(* PLC project PLC107_AO, home PLC107_AO 1 *)
(* stored: creationDateTime 2019-11-13T09:37:45, productRelease 0, modificationDateTime 2020-07-16T10:40:43, version 1 *)

(* Установка режима работы аналогового выхода *)
FUNCTION_BLOCK AOMode
  VAR_INPUT
    Ex : BOOL := FALSE;  (* разрешение на выполнение *)
    AOn : BYTE := 0;  (* номер выхода *)
    M : BYTE := 0;  (* режим работы *)
  END_VAR
  VAR_OUTPUT
    Om : BYTE := 0;  (* режим работы (установленный) *)
    Ok : BYTE := 0;  (* код результата исполнения блока *)
  END_VAR

            {extern void App_AOMode(AOMODE*);App_AOMode(data__);}

          
END_FUNCTION_BLOCK

(* Установка значения нормального аналогового выхода *)
FUNCTION_BLOCK AOVal
  VAR_INPUT
    Ex : BOOL := FALSE;  (* разрешение на выполнение *)
    AOn : BYTE := 0;  (* номер выхода *)
    V : REAL := 0.0;  (* значение *)
  END_VAR
  VAR_OUTPUT
    Ov : REAL := 0.0;  (* значение (установленное) *)
    Ok : BYTE := 0;  (* код результата исполнения блока *)
  END_VAR

            {extern void App_AOVal(AOVAL*);App_AOVal(data__);}

          
END_FUNCTION_BLOCK

(* Установка значения быстрого аналогового выхода *)
FUNCTION_BLOCK AOFast
  VAR_INPUT
    Ex : BOOL := FALSE;  (* разрешение на выполнение *)
    AOn : BYTE := 0;  (* номер выхода *)
    V : REAL := 0.0;  (* значение быстрого выхода *)
  END_VAR
  VAR_OUTPUT
    Ov : REAL := 0.0;  (* значение быстрого выхода (установленное) *)
    Ok : BYTE := 0;  (* код результата исполнения блока *)
  END_VAR

            {extern void App_AOFast(AOFAST*);App_AOFast(data__);}

          
END_FUNCTION_BLOCK

(* Установка безопасного значения аналогового выхода *)
FUNCTION_BLOCK AOSafe
  VAR_INPUT
    Ex : BOOL := FALSE;  (* разрешение на выполнение *)
    Enx : BOOL := FALSE;  (* разрешение быстрого выхода *)
    AOn : BYTE := 0;  (* номер выхода *)
    V : REAL := 0.0;  (* значение быстрого выхода *)
  END_VAR
  VAR_OUTPUT
    Ov : REAL := 0.0;  (* значение быстрого выхода (установленное) *)
    Ow : BOOL := FALSE;  (* разрешение быстрого выхода (установленное) *)
    Ok : BYTE := 0;  (* код результата исполнения блока *)
  END_VAR

            {extern void App_AOSafe(AOSAFE*);App_AOSafe(data__);}

          
END_FUNCTION_BLOCK
